# EPICS autosave request: CARS/iocBoot/iocPINK/auto_positions.req
file "XFM_motor_positions.req",      P=XF:04BM-ES:2:, M=m1
file "XFM_motor_positions.req",      P=XF:04BM-ES:2:, M=m2
file "XFM_motor_positions.req",      P=XF:04BM-ES:2:, M=m3
